// TIA Portal V20 export
FUNCTION_BLOCK "FB_GestionSafetyGate"   // FB202, SCL
{ S7_Optimized_Access := 'TRUE' }
// stored: AutoNumber false, MemoryReserve 100, SetENOAutomatically false
   VAR
      sExtGate { S7_SetPoint := 'True'} : "FB_CmdCylinder";
      sIntGate { S7_SetPoint := 'True'} : "FB_CmdCylinder";
      sExtGateCloseCmd : Bool;
      sExtGateOpenCmd : Bool;
      sIntGateCloseCmd : Bool;
      sIntGateOpenCmd : Bool;
      sJOG_Cmd : Bool;
      sRT_RefCmd : R_TRIG;
      sFT_RefCmd : F_TRIG;
      sExtGateOpenReq : Bool;
      sIntGateOpenReq : Bool;
      sExtGateOpened : Bool;
      sExtGateClosed : Bool;
      sIntGateOpened : Bool;
      sIntGateClosed : Bool;
      sWaitCloseShutterBeforeOpen : Bool;
      sWaitOpenShutterAfterClose : Bool;
      sTimeoutOpenCloseGateTimer : TON_TIME;
      sRT_IntGateOpenbyHMI { S7_SetPoint := 'True'} : R_TRIG;
      sFT_IntGateOpenbyHMI { S7_SetPoint := 'True'} : F_TRIG;
      sRT_ExtGateOpenbyHMI { S7_SetPoint := 'True'} : R_TRIG;
      sFT_ExtGateOpenbyHMI { S7_SetPoint := 'True'} : F_TRIG;
      sRT_ExtGateClose { S7_SetPoint := 'True'} : R_TRIG;
      sRT_ExtGateOpen { S7_SetPoint := 'True'} : R_TRIG;
      sRT_IntGateClose { S7_SetPoint := 'True'} : R_TRIG;
      sRT_IntGateOpen { S7_SetPoint := 'True'} : R_TRIG;
      sInterlockExtGateClose { S7_SetPoint := 'True'} : Bool;
      sInterlockExtGateOpen { S7_SetPoint := 'True'} : Bool;
      sInterlockIntGateClose : Bool;
      sInterlockIntGateOpen : Bool;
   END_VAR
   VAR_TEMP
      tError : Int;
      tCloseExtGate : Bool;
      tOpenExtGate : Bool;
      tCloseIntGate : Bool;
      tOpenIntGate : Bool;
      tSasPosShuttle1 : Real;
      tSasPosShuttle2 : Real;
      tActPosShuttle1 : Real;
      tActPosShuttle2 : Real;
      tDeltaSasShuttle1 : Real;
      tDeltaSasShuttle2 : Real;
      tSynchroMode : Bool;
      tOpenAllGates : Bool;
      tCloseAllGates : Bool;
   END_VAR
   VAR CONSTANT
      TIMEOUT_OPEN_CLOSE_GATE_TIME : Time := T#3s;
   END_VAR
BEGIN
   REGION Description header 
       //==================================================================================
       // POSALUX Swiss SA / (C) Copyright 2025
       //----------------------------------------------------------------------------------
       // Title: Initialization of axis
       // Comment/Function: 
       // Author: Fabien WALDT
       // Engineering: TIA Portal v17
       //----------------------------------------------------------------------------------
       // Change log table:
       // Version  | Date     | Expert in charge | Changes applied
       // ---------|----------|------------------|-----------------------------------------
       // 00.00.01 | 20250509 | WFA              | First released version
       // =================================================================================
   END_REGION

   REGION Reference - Jog Command : Open/Close all Gates
       // Si mode Jog ET Demande reference OU Axe Shuttle selectionné, ouverture SAS Int et Ext
       #sRT_RefCmd(CLK := (("LBP_Chan1".A_Ref OR "MCP1_Out".LEDaxis5 OR "MCP1_Out".LEDaxis6) AND "LBP_ModeGroup".E_JOG)
                  OR "LBP_Chan1".MDyn[45]);     // M45: Open all Gates

       IF #sRT_RefCmd.Q THEN
           #sWaitCloseShutterBeforeOpen := TRUE;
       END_IF;

       IF #sRT_RefCmd.Q THEN
           #tCloseAllGates := FALSE;
       END_IF;

      // #tOpenAllGates := #Wait_close_Shutter_before_open AND ("DB_DataFromSafety".ShutterOpened OR NOT "DB_DataFromSafety".EmergencyStop); WFA A mettre en place quand shutter OK
       #tOpenAllGates := #sWaitCloseShutterBeforeOpen AND (true OR NOT "DB_DataFromSafety".EmergencyStop);

      IF #tOpenAllGates THEN
          #sWaitCloseShutterBeforeOpen := FALSE;
      END_IF;

       #sFT_RefCmd(CLK := (("LBP_Chan1".A_Ref OR "MCP1_Out".LEDaxis5 OR "MCP1_Out".LEDaxis6) AND "LBP_ModeGroup".E_JOG)
                  OR "LBP_Chan1".MDyn[44]);     // M44: Close all Gates

       IF #sFT_RefCmd.Q THEN
           #tCloseAllGates := TRUE;
       END_IF;

       IF #sFT_RefCmd.Q THEN
           #sWaitCloseShutterBeforeOpen := FALSE;
       END_IF;
   END_REGION

   REGION Close Shutter when all gates are open
       IF "LBP_Chan1".MDyn[45] THEN                // M45: Open all Gates
           "DB_DataToSafety".CloseShutter := TRUE;
       END_IF;

       IF "MCP1_In".reset
           OR "LBP_Chan1".MDyn[44] THEN           // M44: Close all Gates
           #sWaitOpenShutterAfterClose := TRUE;
       END_IF;

       IF #sWaitOpenShutterAfterClose AND (NOT "DB_DigitalInputs".sExternalGateLocked.sSWStatus OR NOT "DB_DigitalInputs".sInternalGateLocked.sSWStatus) THEN
           #sWaitOpenShutterAfterClose := FALSE;
           "DB_DataToSafety".CloseShutter := FALSE;
       END_IF;
   END_REGION

   REGION Time Out Gate
       #sTimeoutOpenCloseGateTimer(IN := NOT (("LBP_Chan1".A_Ref OR "MCP1_Out".LEDaxis5 OR "MCP1_Out".LEDaxis6) AND "LBP_ModeGroup".E_JOG) AND (NOT "DB_DigitalInputs".sExternalGateLocked.sSWStatus OR NOT "DB_DigitalInputs".sInternalGateLocked.sSWStatus),
                                   PT := #TIMEOUT_OPEN_CLOSE_GATE_TIME);

       IF #sTimeoutOpenCloseGateTimer.Q THEN
           "LBP_AlarmMsgs".UserA[2].A70UUxx[18]:= TRUE;     // Msg: "700218 - Time out doors SAS int/ext"
       END_IF;
   END_REGION

   REGION Gates management by HMI
       IF "LBP_ModeGroup".E_JOG
           AND NOT "LBP_Chan1".A_Ref
           AND NOT "MCP1_Out".LEDaxis5
           AND NOT "MCP1_Out".LEDaxis6 THEN
           #sRT_IntGateOpenbyHMI(CLK := "DB_HMICmd".IntGateOpenReq,
                                 Q => "DB_HMICmd".IntGateOpenCmd);

           #sFT_IntGateOpenbyHMI(CLK := "DB_HMICmd".IntGateOpenReq,
                                 Q => "DB_HMICmd".IntGateCloseCmd);

           #sRT_ExtGateOpenbyHMI(CLK := "DB_HMICmd".ExtGateOpenReq,
                                 Q => "DB_HMICmd".ExtGateOpenCmd);

           #sFT_ExtGateOpenbyHMI(CLK := "DB_HMICmd".ExtGateOpenReq,
                                 Q => "DB_HMICmd".ExtGateCloseCmd);
       END_IF;
   END_REGION

   REGION Syncro Mode
       #tSynchroMode := "DB_LoaderShuttle1".sMain.sInterface.SequenceRun
       AND "DB_LoaderShuttle2".sMain.sInterface.SequenceRun
       AND (("DB_LoaderShuttle1".sShuttleInt.oExtGateOpenReq AND "DB_LoaderShuttle2".sShuttlePosSas)
         OR ("DB_LoaderShuttle1".sShuttleInt.oIntGateOpenReq AND "DB_LoaderShuttle2".sShuttlePosInt)
         OR ("DB_LoaderShuttle1".sShuttleExt.oExtGateOpenReq AND "DB_LoaderShuttle2".sShuttlePosExt)
         OR ("DB_LoaderShuttle1".sShuttleExt.oIntGateOpenReq AND "DB_LoaderShuttle2".sShuttlePosSas)
         OR ("DB_LoaderShuttle2".sShuttleInt.oExtGateOpenReq AND "DB_LoaderShuttle1".sShuttlePosSas)
         OR ("DB_LoaderShuttle2".sShuttleInt.oIntGateOpenReq AND "DB_LoaderShuttle1".sShuttlePosInt)
         OR ("DB_LoaderShuttle2".sShuttleExt.oExtGateOpenReq AND "DB_LoaderShuttle1".sShuttlePosExt)
         OR ("DB_LoaderShuttle2".sShuttleExt.oIntGateOpenReq AND "DB_LoaderShuttle1".sShuttlePosSas));
   END_REGION

   REGION Gates management by M Codes - PLC Sequence
       IF #tCloseAllGates THEN
           #sExtGateOpenReq := FALSE;
           #sIntGateOpenReq := FALSE;
       END_IF;

       // External Gate
       IF "LBP_Chan1".MDyn[46]                         // M46: Closing External Gate (Not in ISO Code)
           OR "DB_LoaderShuttle1".oExtGateCloseReq     // Closure External Gate request from Shuttle 1
           OR "DB_LoaderShuttle2".oExtGateCloseReq     // Closure External Gate request from Shuttle 2
           OR "DB_HMICmd".ExtGateCloseCmd THEN         // Closure External Gate request from HMI
               #sExtGateOpenReq := FALSE;
       END_IF;

       IF "LBP_Chan1".MDyn[47]                                                                                                                            // M47: Opening External Gate (Not in ISO Code)
           OR (("DB_LoaderShuttle1".oExtGateOpenReq OR "DB_LoaderShuttle2".oExtGateOpenReq) AND NOT "DB_LoaderMain".sSynchroMode AND NOT #tSynchroMode)   // Opening External Gate request from Shuttle 1 or 2 (Only one Shuttle sequence is running)
           OR (("DB_LoaderShuttle1".oExtGateOpenReq AND "DB_LoaderShuttle2".oExtGateOpenReq) AND ("DB_LoaderMain".sSynchroMode OR #tSynchroMode))         // Opening External Gate request from Shuttle 1 and 2 (both Shuttle sequence are running)
           OR "DB_HMICmd".ExtGateOpenCmd                                                                                                                  // Opening External Gate request from HMI
           OR (("LBP_Chan1".A_Ref OR "MCP1_Out".LEDaxis5 OR "MCP1_Out".LEDaxis6) AND "LBP_ModeGroup".E_JOG) THEN                                          // Opening External Gate request from Mode Group
               #sExtGateOpenReq := TRUE;
       END_IF;

       #sRT_ExtGateClose(CLK:=NOT  #sExtGateOpenReq AND NOT #sInterlockExtGateClose,
                             Q=> #tCloseExtGate);

       #sRT_ExtGateOpen(CLK := #sExtGateOpenReq AND NOT #sInterlockExtGateOpen,
                            Q => #tOpenExtGate);

        // Internal Gate
       IF "LBP_Chan1".MDyn[48]                         // M48: Closing Internal Gate (Not in ISO Code)
           OR "DB_LoaderShuttle1".oIntGateCloseReq     // Closure Internal Gate request from Shuttle 1
           OR "DB_LoaderShuttle2".oIntGateCloseReq     // Closure Internal Gate request from Shuttle 2
           OR "DB_HMICmd".IntGateCloseCmd THEN         // Closure External Gate request from HMI
               #sIntGateOpenReq := FALSE;
       END_IF;

       IF "LBP_Chan1".MDyn[49]                                                                                                                            // M49: Opening Internal Gate (Not in ISO Code)
           OR (("DB_LoaderShuttle1".oIntGateOpenReq OR "DB_LoaderShuttle2".oIntGateOpenReq) AND NOT "DB_LoaderMain".sSynchroMode AND NOT #tSynchroMode)   // Opening Internal Gate request from Shuttle 1 or 2 (Only one Shuttle sequence is running)
           OR (("DB_LoaderShuttle1".oIntGateOpenReq AND "DB_LoaderShuttle2".oIntGateOpenReq) AND ("DB_LoaderMain".sSynchroMode OR #tSynchroMode))         // Opening Internal Gate request from Shuttle 1 and 2 (both Shuttle sequence are running)
           OR "DB_HMICmd".IntGateOpenCmd                                                                                                                  // Opening External Gate request from HMI
           OR (("LBP_Chan1".A_Ref OR "MCP1_Out".LEDaxis5 OR "MCP1_Out".LEDaxis6) AND "LBP_ModeGroup".E_JOG) THEN                                          // Opening External Gate request from Mode Group
           #sIntGateOpenReq := TRUE;
       END_IF;

       #sRT_IntGateClose(CLK := NOT #sIntGateOpenReq AND NOT #sInterlockIntGateClose,
                          Q => #tCloseIntGate);

        #sRT_IntGateOpen(CLK := #sIntGateOpenReq AND NOT #sInterlockIntGateOpen,
                          Q => #tOpenIntGate);
    END_REGION

    REGION Interlocks
        #sInterlockExtGateOpen := NOT #sIntGateClosed OR #sIntGateOpenReq;
        #sInterlockIntGateOpen := NOT #sExtGateClosed OR #sExtGateOpenReq;

        #sInterlockExtGateClose := ("DB_AxisPosition".sAxis05_U1."$AA_IM" >= "DB_AxisPosMachinePLC".Axis_U1.ExtGateExt
        AND "DB_AxisPosition".sAxis05_U1."$AA_IM" <= "DB_AxisPosMachinePLC".Axis_U1.IntGateExt)
        OR ("DB_AxisPosition".sAxis06_U2."$AA_IM" >= "DB_AxisPosMachinePLC".Axis_U2.ExtGateExt
        AND "DB_AxisPosition".sAxis06_U2."$AA_IM" <= "DB_AxisPosMachinePLC".Axis_U2.IntGateExt);

        #sInterlockIntGateClose := ("DB_AxisPosition".sAxis05_U1."$AA_IM" >= "DB_AxisPosMachinePLC".Axis_U1.ExtGateInt
        AND "DB_AxisPosition".sAxis05_U1."$AA_IM" <= "DB_AxisPosMachinePLC".Axis_U1.IntGateInt)
        OR ("DB_AxisPosition".sAxis06_U2."$AA_IM" >= "DB_AxisPosMachinePLC".Axis_U2.ExtGateInt
        AND "DB_AxisPosition".sAxis06_U2."$AA_IM" <= "DB_AxisPosMachinePLC".Axis_U2.IntGateInt);
    END_REGION

    REGION External Gate Command
        #sExtGateCloseCmd := (#tCloseAllGates OR #tCloseExtGate) AND NOT #sInterlockExtGateClose;
        #sExtGateOpenCmd := #tOpenAllGates OR (#tOpenExtGate AND NOT #sInterlockExtGateOpen);
    END_REGION

    REGION Internal Gate Command
        #sIntGateCloseCmd := (#tCloseAllGates OR #tCloseIntGate) AND NOT #sInterlockIntGateClose;
        #sIntGateOpenCmd := #tOpenAllGates OR (#tOpenIntGate AND NOT #sInterlockIntGateOpen);
    END_REGION 

    REGION External Gate
        #sExtGate(iEMinus := "DB_DigitalInputs".sExternalGateLocked.sSWStatus,
                  iEPlus := "DB_DigitalInputs".sExternalGateOpened.sSWStatus,
                  iMinusCmd := #sExtGateCloseCmd,
                  iPlusCmd := #sExtGateOpenCmd,
                  iJOGCmd := #sJOG_Cmd,
                  iMonitorTime := T#8s,
                  oErrorCode => #tError,
                  ioQMinus := "DB_DigitalOutputs".sExternalGateClosing.sSWStatus,
                  ioQPlus := "DB_DigitalOutputs".sExternalGateOpening.sSWStatus);

        CASE #tError OF
            1:
                "LBP_AlarmMsgs".UserA[2].A70UUxx[21] := TRUE;  // Msg: "700221 - Time out door ext. SAS closing"
            2:
                "LBP_AlarmMsgs".UserA[2].A70UUxx[19] := TRUE;  // Msg: "700219 - Time out door ext. SAS opening"
        END_CASE;
    END_REGION ;

    REGION Internal Gate
        #sIntGate(iEMinus:= "DB_DigitalInputs".sInternalGateLocked.sSWStatus,
                  iEPlus:=  "DB_DigitalInputs".sInternalGateOpened.sSWStatus,
                  iMinusCmd:=#sIntGateCloseCmd,
                  iPlusCmd:=#sIntGateOpenCmd,
                  iJOGCmd:=#sJOG_Cmd,
                  iMonitorTime:=T#8s,
                  oErrorCode=>#tError,
                  ioQMinus:="DB_DigitalOutputs".sInternalGateClosing.sSWStatus,
                  ioQPlus:="DB_DigitalOutputs".sInternalGateOpening.sSWStatus);

        CASE #tError OF
            1:
               "LBP_AlarmMsgs".UserA[2].A70UUxx[22] := TRUE;  // Msg: "700222 - Time out door int. SAS closing" (WFA à corriger)
            2:
               "LBP_AlarmMsgs".UserA[2].A70UUxx[20] := TRUE;  // Msg: "700220 - Time out door int. SAS opening" (WFA à corriger)
        END_CASE;
    END_REGION ;

    REGION Gates Status 
        // External Gate Closed
        #sExtGateClosed := "DB_DigitalInputs".sExternalGateLocked.sSWStatus
        AND NOT "DB_DigitalInputs".sExternalGateOpened.sSWStatus;

        // External Gate Open
        #sExtGateOpened := NOT "DB_DigitalInputs".sExternalGateLocked.sSWStatus
        AND "DB_DigitalInputs".sExternalGateOpened.sSWStatus;

        // Internal Gate Closed
        #sIntGateClosed := "DB_DigitalInputs".sInternalGateLocked.sSWStatus
        AND NOT "DB_DigitalInputs".sInternalGateOpened.sSWStatus;

        // Internal Gate Open
        #sIntGateOpened := NOT "DB_DigitalInputs".sInternalGateLocked.sSWStatus
        AND "DB_DigitalInputs".sInternalGateOpened.sSWStatus;
    END_REGION ;
END_FUNCTION_BLOCK
